FUNCTION_BLOCK ConveyorCTLServer (* Basic Function Block Type *)
  (* Standard: 61499-2 *)
  (* Version 0.2, 2003-12-04, JHC, Rockwell Automation, Renamed for better indexing. *)
  (* Version 0.1, 2002-11-05, JHC, Rockwell Automation, Corrected missing ST element in Algorithm REQ. *)
  (* Version 0.0, 2000-05-30, JHC, Rockwell Automation *)
  (* Compiler header: package fb.rt.cs725; *)
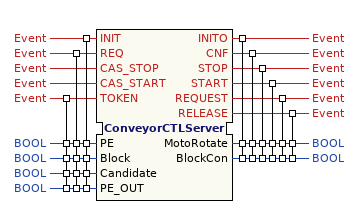
  EVENT_INPUT
    INIT WITH PE, Block, Candidate, PE_OUT; (* Initialization Request *)
    REQ WITH PE, Block, Candidate, PE_OUT; (* Normal Execution Request *)
    CAS_STOP;
    CAS_START;
    TOKEN WITH PE, Block, Candidate, PE_OUT;
  END_EVENT
  EVENT_OUTPUT
    INITO WITH MotoRotate, BlockCon; (* Initialization Confirm *)
    CNF WITH MotoRotate, BlockCon; (* Execution Confirmation *)
    STOP WITH MotoRotate, BlockCon;
    START WITH MotoRotate, BlockCon;
    REQUEST WITH MotoRotate, BlockCon;
    RELEASE WITH BlockCon, MotoRotate;
  END_EVENT
  VAR_INPUT
    PE : BOOL; (* Input event qualifier *)
    Block : BOOL;
    Candidate : BOOL;
    PE_OUT : BOOL;
  END_VAR
  VAR_OUTPUT
    MotoRotate : BOOL; (* Output event qualifier *)
    BlockCon : BOOL;
  END_VAR
  VAR
    lastPE : BOOL := 1;
    lastBlock : BOOL := 0;
  END_VAR
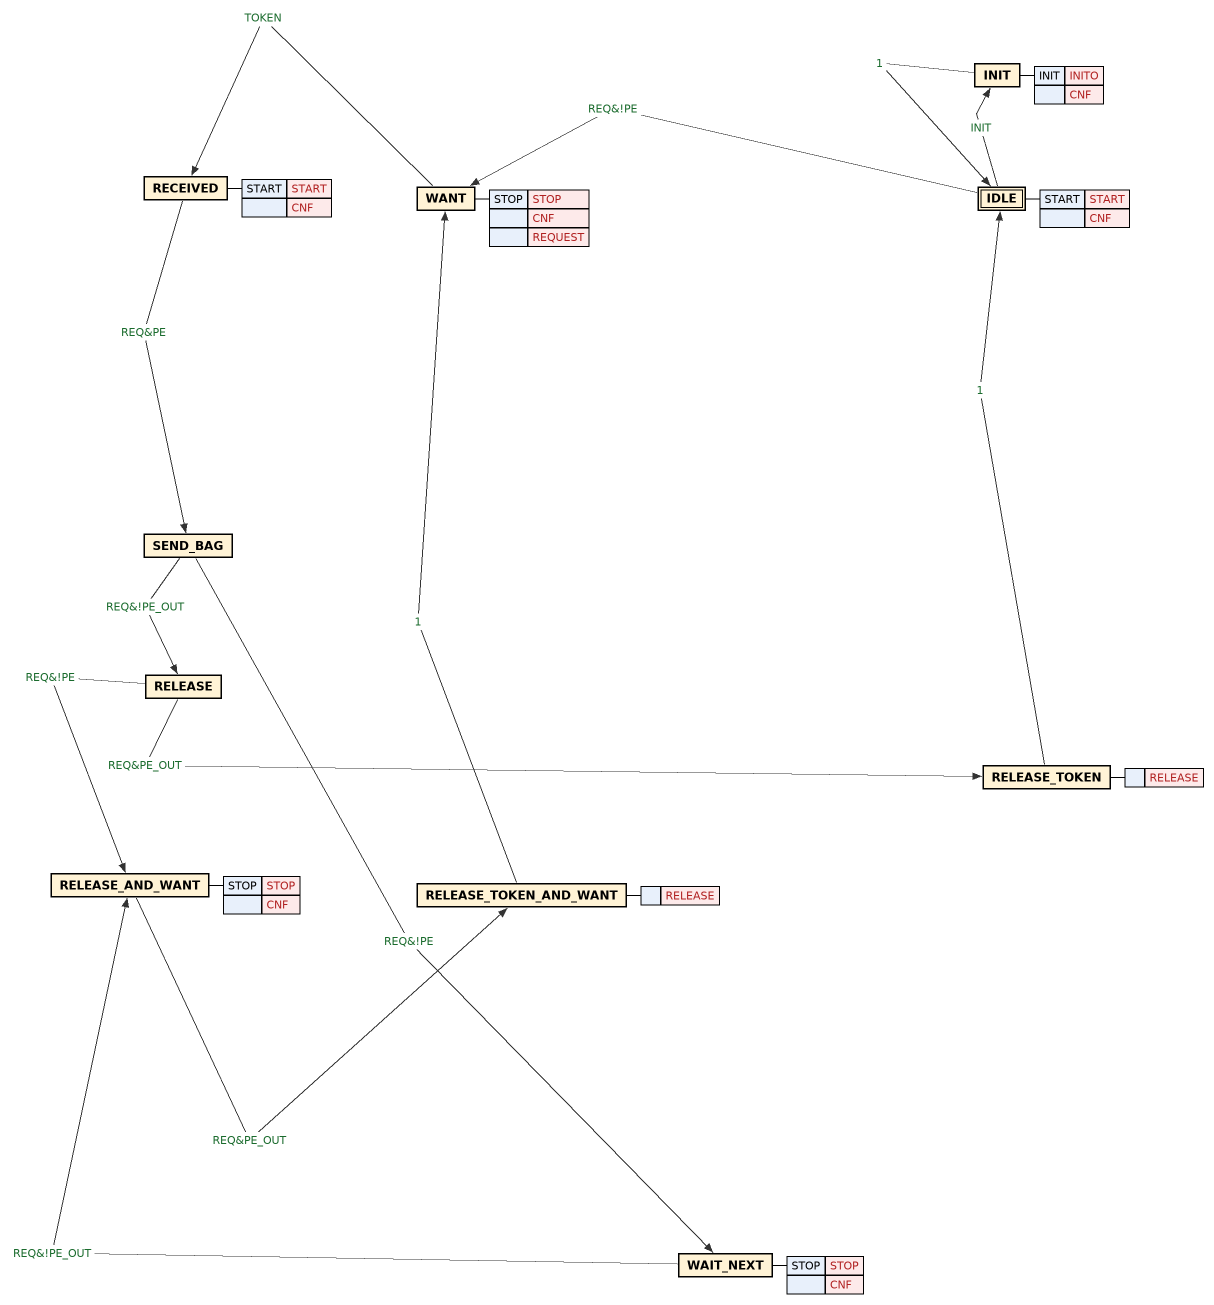
  EC_STATES
    IDLE : START -> START, -> CNF; (* Initial State *)
    INIT : INIT -> INITO, -> CNF; (* Initialization *)
    WANT : STOP -> STOP, -> CNF, -> REQUEST;
    RECEIVED : START -> START, -> CNF;
    WAIT_NEXT : STOP -> STOP, -> CNF;
    SEND_BAG;
    RELEASE;
    RELEASE_AND_WANT : STOP -> STOP, -> CNF;
    RELEASE_TOKEN : -> RELEASE;
    RELEASE_TOKEN_AND_WANT : -> RELEASE;
  END_STATES
  EC_TRANSITIONS
    IDLE TO INIT := INIT;
    INIT TO IDLE := 1;
    WANT TO RECEIVED := TOKEN;
    RECEIVED TO SEND_BAG := REQ&PE;
    SEND_BAG TO WAIT_NEXT := REQ&!PE;
    WAIT_NEXT TO RELEASE_AND_WANT := REQ&!PE_OUT;
    SEND_BAG TO RELEASE := REQ&!PE_OUT;
    RELEASE_TOKEN TO IDLE := 1;
    RELEASE TO RELEASE_TOKEN := REQ&PE_OUT;
    RELEASE_TOKEN_AND_WANT TO WANT := 1;
    RELEASE_AND_WANT TO RELEASE_TOKEN_AND_WANT := REQ&PE_OUT;
    RELEASE TO RELEASE_AND_WANT := REQ&!PE;
    IDLE TO WANT := REQ&!PE;
  END_TRANSITIONS
  ALGORITHM INIT IN ST: (* Initialization algorithm *)
MotoRotate := TRUE;
Block := FALSE;

System.out.println(this + " " + MotoRotate);
System.out.println(MotoRotate);
  END_ALGORITHM
  ALGORITHM REQ IN ST: (* Normally executed algorithm *)
System.out.println(this +  " -> Candidate" + Candidate);
IF Candidate THEN
IF lastPE !:= PE THEN
IF NOT PE THEN
BlockCon:= TRUE;
System.out.println("BlockCon = true");
ELSE
BlockCon:=FALSE;
System.out.println("BlockCon = false");
END_IF
lastPE := PE;
END_IF
IF lastBlock !:= Block THEN
IF Block THEN
STOP.serviceEvent(this);
MotoRotate := FALSE;
System.out.println("Cas Stop");
ELSE
START.serviceEvent(this);
MotoRotate := TRUE;
System.out.println("Cas Start");
END_IF
lastBlock := Block;
END_IF
END_IF
  END_ALGORITHM
  ALGORITHM START IN ST:
MotoRotate:=TRUE;
System.out.println(this + " Start " + MotoRotate);

System.out.println("Start " + MotoRotate);
  END_ALGORITHM
  ALGORITHM STOP IN ST:
MotoRotate := FALSE;
System.out.println(this + " Stop " + MotoRotate);

System.out.println("Stop " + MotoRotate);
  END_ALGORITHM
END_FUNCTION_BLOCK
